% RSLogix 500 project A&B TEST11.RSS, saved by version 8.30.00.16 %
PROJECT "TEST1"    % processor: MicroLogix 1000 %

PROGRAM FILES
  LAD 2 "MAIN_PROG"  7 rungs
  LAD 3 "USER_FAULT"  1 rungs
  LAD 4 "HSC_INT"  1 rungs
  LAD 5 "STI_INT"  1 rungs
  LAD 6, 7, 8, 9, 10, 11, 12, 13, 14, 15, 16: only END

DATA FILES
  O0 OUTPUT  1 elements
  I1 INPUT  2 elements
  S2 STATUS  33 elements
  B3 BINARY  32 elements
  T4 TIMER  40 elements
  C5 COUNTER  32 elements
  R6 CONTROL  16 elements
  N7 INTEGER  105 elements

LADDER 2 "MAIN_PROG"
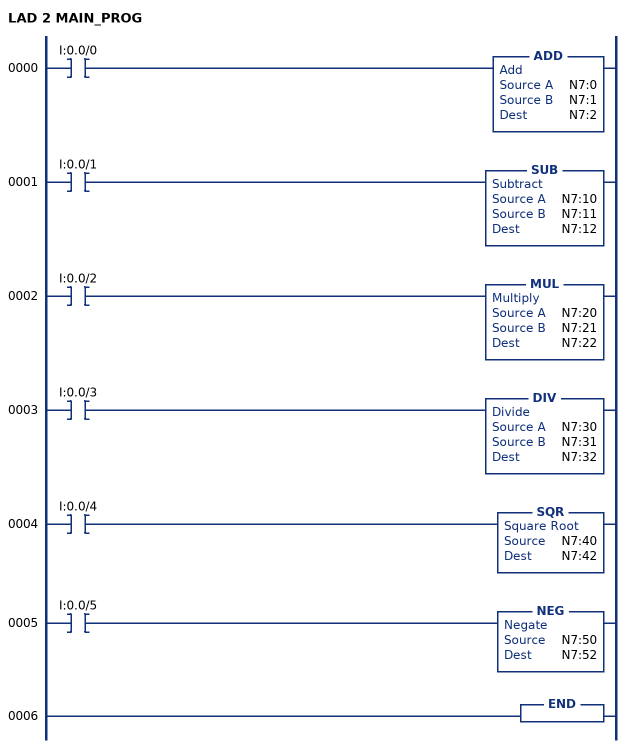
% Rung: 0 %
SOR XIC I:0.0/0 ADD N7:0 N7:1 N7:2 EOR
% Rung: 1 %
SOR XIC I:0.0/1 SUB N7:10 N7:11 N7:12 EOR
% Rung: 2 %
SOR XIC I:0.0/2 MUL N7:20 N7:21 N7:22 EOR
% Rung: 3 %
SOR XIC I:0.0/3 DIV N7:30 N7:31 N7:32 EOR
% Rung: 4 %
SOR XIC I:0.0/4 SQR N7:40 N7:42 EOR
% Rung: 5 %
SOR XIC I:0.0/5 NEG N7:50 N7:52 EOR
% Rung: 6 %
SOR END EOR

DATA TABLE (non-zero values as saved)
DATA T4
% .PRE .ACC %
% T4:0 % 15 0
DATA C5
% .PRE .ACC %
% C5:0 % 5 0
